# EPICS substitutions: iocs/MC06/db/SAI_EncoderLoss.substitutions
file /opt/epics/modules/SAI/db/SAI_EncoderLoss.template {
pattern {	P,		R,	AXIS,	SCAN, 		ASYNPORT, 	VARSTS, VARCLR}
        { 	"XF:06BM-BI",		"{FS:03-Ax:",	"Y}Mtr","1 second",	"pmac",		"M181",	"M901"}
        { 	"XF:06BM-BI",		"{BPM:1-Ax:",	"Y}Mtr","1 second",	"pmac",		"M281",	"M901"}
        { 	"XF:06BM-BI",		"{BCT-Ax:",	"Y}Mtr","1 second",	"pmac",		"M381",	"M901"}
        { 	"XF:06BM-BI",		"{Fltr:01-Ax:",	"Y}Mtr","1 second",	"pmac",		"M481",	"M901"}
        { 	"XF:06BM-BI",		"{Slt:02-Ax:",	"O}Mtr","1 second",	"pmac",		"M581",	"M901"}
        { 	"XF:06BM-BI",		"{Slt:02-Ax:",	"I}Mtr","1 second",	"pmac",		"M681",	"M901"}
        { 	"XF:06BM-BI",		"{Slt:02-Ax:",	"T}Mtr","1 second",	"pmac",		"M781",	"M901"}
        { 	"XF:06BM-BI",		"{Slt:02-Ax:",	"B}Mtr","1 second",	"pmac",		"M881",	"M901"}
}

#EOF
